(* CODESYS project JobManagement.library
   Company: Bekchoff Automation K.K.
   DocFormat: reStructuredText
   DefaultNamespace: jobmgmt
   Version: 1.0.0.1
   Placeholder: JobManagementFramework
   Author: Takashi Ichihashi
   Title: JobManagementFramework

Project tree, tasks and I/O mapping:
  libraries: Tc2_Standard, * (Beckhoff Automation GmbH); Tc2_System, * (Beckhoff Automation GmbH); Tc2_Utilities, * (Beckhoff Automation GmbH); Tc3_Module, * (Beckhoff Automation GmbH); VisuSymbols, 3.5.10.0 (System)
  DUTs/
    data type ContainerType
    data type E_ErrorId
    data type E_FutureExecutionState
    data type ST_MotionData
  GVLs/
    global variables GVL
    global variables ParamFuturesLib
  POUs/
    model/
      activities/
        function block FB_observer [ST]: subscribe_job_directory, subscribe_job_event
        function block FutureCounterBlink [ST]: abort, counter, error_reset, error_test, execute, init, nErrorID, quit, set_options, set_parameter
        function block FutureCounterBlinkCreator [ST]: create_future, destroy_future, set_options, set_parameter
        function block FutureTimerBlink [ST]: abort, error_reset, error_test, execute, init, nErrorID, quit, set_options, set_parameter
        function block FutureTimerBlinkCreator [ST]: create_future, destroy_future, set_options, set_parameter
      library/
        function block FB_AbstructContainer [ST]: _append_job, _index_generator_, abort, append_job, auto_start, continuous_mode, create_container, create_job, each_executor, error_reset, execute, executor, future_name, init, nErrorID, num_of_jobs, quit, reset, resume, spawn_job, start, state
        function block FB_AbstructFuture [ST]: abort, error_reset, execute, executor, future_name, init, nErrorID, quit, state
        function block FB_BatchJobContainer [ST]: _append_job, _index_generator_, abort, execute, init, quit, resume, start
        function block FB_BatchJobContainerCreator [ST]: create_future, destroy_future
        function block FB_Executor [ST]: abort, busy, children, continuous_mode, create_container, create_future, current_state, done, error_reset, execute, future, future_creator, id, init, job_event_reporter, last_state, nErrorID, parent_executor, persistent_job, quit, ready, reset, resume, start, uid, upstream_aborting
        function block FB_ExecutorTreeSearch [ST]: search, subscriber
        function block FB_ParallelJobContainer [ST]: _append_job, _index_generator_, abort, execute, init, quit, start
        function block FB_ParallelJobContainerCreator [ST]: create_future, destroy_future
        function block FB_ParallelQueueJobContainer [ST]: _append_job, _index_generator_, abort, execute, init, start
        function block FB_ParallelQueueJobContainerCreator [ST]: create_future, destroy_future
        function block FB_QueueJobContainer [ST]: _append_job, _index_generator_, abort, dequeue, execute, init, start
        function block FB_QueueJobContainerCreator [ST]: create_future, destroy_future
        interface InterfaceContainer: _index_generator_, append_job, auto_start, continuous_mode, create_container, create_job, each_executor, num_of_jobs, reset, resume, spawn_job, start
        interface InterfaceFuture: abort, error_reset, execute, executor, future_name, init, nErrorID, quit, state
        interface InterfaceObserver: subscribe_job_directory, subscribe_job_event
        interface InterfaceTaskCreator: create_future, destroy_future
    program MAIN [ST]
  VISUs/
    visualisation Visualization
    visualisation Visualization_1
  text list GlobalTextList
*)

// DUTs/ContainerType
{attribute 'qualified_only'}
{attribute 'strict'}
TYPE ContainerType :
(
	BATCH := 0,
	PARALLEL,
	QUEUE,
	PARALLEL_QUEUE
);
END_TYPE

// DUTs/E_ErrorId
{attribute 'qualified_only'}
{attribute 'strict'}
TYPE E_ErrorId :
(
	PASSIVE_ABORT := 16#FFFFFFFF,
	NOT_CONTAINER := 16#FFFFFFFE
) UDINT;
END_TYPE

// DUTs/E_FutureExecutionState
{attribute 'qualified_only'}
{attribute 'strict'}
{attribute 'to_string'}
TYPE E_FutureExecutionState :
(
	idle := 0,
	init,
	wait_for_process,
	process,
	abort,
	pause,
	quit,
	finish
);
END_TYPE

// DUTs/ST_MotionData
TYPE ST_MotionData :
STRUCT
	name: STRING;
	position: LREAL;
	speed: LREAL;
	accel: LREAL;
END_STRUCT
END_TYPE

// GVLs/GVL
{attribute 'qualified_only'}
VAR_GLOBAL
	batch_job_container_creator : FB_BatchJobContainerCreator;
	parallel_job_container_creator : FB_ParallelJobContainerCreator;
	queue_job_container_creator : FB_QueueJobContainerCreator;
	parallel_queue_job_container_creator : FB_ParallelQueueJobContainerCreator;
END_VAR

// GVLs/ParamFuturesLib
{attribute 'qualified_only'}
VAR_GLOBAL CONSTANT
	MAX_TASK_NUM : UINT := 1000; // Number of max jobs in job container object.
	MAX_STRING_LENGTH : UDINT := 255; // Max string length of task name.
END_VAR

// POUs/model/activities/FB_observer
FUNCTION_BLOCK FB_observer IMPLEMENTS InterfaceObserver
VAR_INPUT
END_VAR
VAR_OUTPUT
	{attribute 'TcEncoding':='UTF-8'}
	text : T_MAXSTRING;
END_VAR
VAR
END_VAR

METHOD subscribe_job_directory : BOOL
VAR_INPUT
	executor	: REFERENCE TO FB_Executor;
END_VAR
VAR
	job_log : STRING;
END_VAR
IF __ISVALIDREF(executor) THEN

	job_log := CONCAT(job_log, 'JOB STRUCTURE');
	IF executor.future <> 0 THEN
		job_log := CONCAT(job_log, '/ FUTURE_NAME : ');
		job_log := CONCAT(job_log, executor.future.future_name);
		job_log := CONCAT(job_log, ', ');	
	END_IF
	job_log := CONCAT(job_log, 'JOB_ID : ');
	job_log := CONCAT(job_log, executor.uid);

	ADSLOGSTR(msgCtrlMask := ADSLOG_MSGTYPE_LOG, msgFmtStr := job_log, strArg := '');
END_IF
END_METHOD

METHOD subscribe_job_event : BOOL
VAR_INPUT
	subject		: T_MaxString;
	old_state	: E_FutureExecutionState;
	new_state	: E_FutureExecutionState;
	record_time	: Tc2_Utilities.T_FILETIME64;
	executor	: REFERENCE TO FB_Executor;
END_VAR
VAR_INST
	fb_timezone_info : FB_GetTimeZoneInformation := (bExecute := TRUE);
END_VAR
VAR
	last_state : STRING;
	current_state : STRING;
	container : InterfaceContainer;
	num_of_jobs : UINT;
END_VAR
last_state := TO_STRING(old_state);
current_state := TO_STRING(new_state);

IF __QUERYINTERFACE(executor.future, container) THEN
	num_of_jobs := container.num_of_jobs;
ELSE
	num_of_jobs := 1;
END_IF


IF __ISVALIDREF(executor) THEN
	fb_timezone_info();
	text := FILETIME64_TO_ISO8601(fileTime := record_time, nBias := DINT_TO_INT(fb_timezone_info.tzInfo.bias), bUTC := TRUE,nPrecision := 6);
	text := CONCAT(text, '	');
	text := CONCAT(text, subject);
	text := CONCAT(text, '	');
	text := CONCAT(text, TO_STRING(current_state));
	text := CONCAT(text, '	');
	text := CONCAT(text, TO_STRING(executor.nErrorID));
	text := CONCAT(text, '		');
	text := CONCAT(text, executor.future.future_name);
	text := CONCAT(text, '		');
	text := CONCAT(text, executor.uid);
	text := CONCAT(text, '		');
	text := CONCAT(text, TO_STRING(num_of_jobs));
	
	
	ADSLOGSTR(msgCtrlMask := ADSLOG_MSGTYPE_LOG,
 			 msgFmtStr := text, 
			strArg := '');	
END_IF

subscribe_job_event := TRUE;
END_METHOD

END_FUNCTION_BLOCK

// POUs/model/library/InterfaceObserver
INTERFACE InterfaceObserver

METHOD subscribe_job_directory : BOOL
VAR_INPUT
	executor: REFERENCE TO FB_Executor; // Represent reference to subscribed job object
END_VAR
END_METHOD

METHOD subscribe_job_event : BOOL
VAR_INPUT
	subject	  : T_MaxString;	// Subject text of event
	old_state : E_FutureExecutionState; // Job state before transition.
	new_state : E_FutureExecutionState; // Job state after transition.
	record_time	: T_FILETIME64; // File-time at the time of transition.
	executor	: REFERENCE TO FB_Executor; // Reference to job instance of which transition occurs.
END_VAR
END_METHOD

END_INTERFACE

// POUs/model/library/FB_Executor
{attribute 'enable_dynamic_creation'}
FUNCTION_BLOCK FB_Executor
VAR_INPUT
END_VAR
VAR_OUTPUT
END_VAR
VAR
	{attribute 'TcEncoding':='UTF-8'}
	_id : T_MaxString;
	_done : BOOL;
	_start : BOOL;
	_resume : BOOL;
	_passive_abort : BOOL;
	_quit : BOOL;
	_upstream_aborting : BOOL := TRUE;
	 {attribute 'TcAnalytics'}
	 _state :E_FutureExecutionState := E_FutureExecutionState.idle;
	_last_state  :E_FutureExecutionState;
	_error_id : UDINT;
	_aborting :BOOL;
	_quitting :BOOL;
	_interface_container : InterfaceContainer := 0;
	_job_event_reporter: InterfaceObserver;
	_future_creator : InterfaceTaskCreator;
	_future : InterfaceFuture;
	_parent_executor : REFERENCE TO FB_Executor REF= 0;
	_persistent_job : BOOL;
END_VAR

(*abort method

*)
METHOD abort : BOOL // Return TRUE if finish.
VAR_INPUT
END_VAR
IF _state = E_FutureExecutionState.init OR
   _state = E_FutureExecutionState.process OR
   _state = E_FutureExecutionState.quit THEN
   	_start := FALSE;
	_passive_abort := TRUE;	
	THIS^.execute();
END_IF

IF 	_passive_abort AND _state = E_FutureExecutionState.abort THEN
	abort := NOT _aborting;
ELSE
	abort := TRUE;
END_IF
END_METHOD

PROPERTY busy : BOOL
GET
busy := (	_state = E_FutureExecutionState.init OR	
			_state = E_FutureExecutionState.process OR 
			_state = E_FutureExecutionState.quit
		);
END_GET
END_PROPERTY

PROPERTY children : InterfaceContainer // Accesser for interface pointer to child container instance.
GET
children := _interface_container;
END_GET
END_PROPERTY

PROPERTY continuous_mode : bool // Make true if keep executing state after all jobs be finished.
SET
IF _future <> 0 THEN
	IF __QUERYINTERFACE(_future, _interface_container) THEN
		_interface_container.continuous_mode := continuous_mode;
	END_IF	
END_IF
END_SET
END_PROPERTY

METHOD create_container : InterfaceContainer // Make container object onto child.
VAR_INPUT
	container_type : ContainerType; // specify container type
	name: STRING;	// specify future name
END_VAR
VAR
	delete_existing_container : BOOL;
	created_future : InterfaceFuture;
END_VAR
IF _interface_container <> 0 THEN
 	IF _interface_container.reset(FALSE) THEN
		delete_existing_container := TRUE;
	ELSE
		delete_existing_container := FALSE;
	END_IF
ELSE
	delete_existing_container := TRUE;
END_IF

IF delete_existing_container THEN
	CASE container_type OF
		ContainerType.BATCH:
			created_future := create_future(GVL.batch_job_container_creator, name);
			created_future.executor.persistent_job := FALSE;
		ContainerType.PARALLEL:
			created_future := create_future(GVL.parallel_job_container_creator, name);
			created_future.executor.persistent_job := FALSE;
		ContainerType.QUEUE:
			created_future := create_future(GVL.queue_job_container_creator, name);
			created_future.executor.persistent_job := TRUE;
		ContainerType.PARALLEL_QUEUE:
			created_future := create_future(GVL.parallel_queue_job_container_creator, name);
			created_future.executor.persistent_job := TRUE;
	END_CASE
	THIS^.init();
	create_container := THIS^.children;
END_IF
END_METHOD

METHOD create_future : InterfaceFuture // Create future dynamically.
VAR_INPUT
	creator : InterfaceTaskCreator; // Specify creator object by which Interface Task Creator implemented.
	future_name: STRING; // Spcfigy future name.
END_VAR
_future_creator := creator;
IF _future_creator <> 0 THEN
	THIS^.future := creator.create_future(future_name);
END_IF
create_future := _future;
END_METHOD

{attribute 'OPC.UA.DA.Property' := '1'}
{attribute 'monitoring' := 'call'}
{attribute 'OPC.UA.DA.Description' := 'Current state of this executor object.'}
PROPERTY current_state : E_FutureExecutionState // Get current job state
GET
current_state := _state;
END_GET
END_PROPERTY

PROPERTY done : BOOL // Present true if process be finished.
GET
done := _done;
END_GET
END_PROPERTY

METHOD error_reset : BOOL
VAR_INPUT
END_VAR
IF _future <> 0 THEN
	IF _future.error_reset() THEN
		error_reset := TRUE;
		IF _job_event_reporter <> 0 THEN
			_job_event_reporter.subscribe_job_event(
						subject := 'ERROR_RESET',
						old_state := _last_state,
						new_state := _state,
						record_time := F_GetSystemTime(),
						executor := THIS^
				);
		END_IF
	ELSE
		error_reset := FALSE;
	END_IF
	_error_id := _future.nErrorID;
ELSE
	_error_id := 0;
	error_reset := TRUE;
END_IF
END_METHOD

METHOD execute : BOOL // Execute future process and return TRUE if all task are finished.
VAR_INST
	_state_mem :E_FutureExecutionState;
	_logging :BOOL;
	delay : TIME := T#3S;
	sleep : TON;
END_VAR
VAR
	_executor : REFERENCE TO FB_Executor;
	start_all_children : BOOL;
	exe: INT;
END_VAR
IF _future = 0 THEN
	execute := TRUE;
	RETURN;
ELSE
	execute := FALSE;
END_IF

IF _passive_abort THEN
	_state := E_FutureExecutionState.abort;
	IF _error_id = 0 THEN
		_error_id := E_ErrorId.PASSIVE_ABORT;
	END_IF
	_passive_abort := FALSE;
END_IF

IF _quit THEN
	_state := E_FutureExecutionState.quit;
END_IF
_quit := FALSE;

CASE _state OF
	E_FutureExecutionState.idle:
		ADSLOGSTR(msgCtrlMask := ADSLOG_MSGTYPE_LOG, msgFmtStr := TO_STRING(_future.state), strArg := '');
		IF _future.state = E_FutureExecutionState.idle OR 
			_future.state = E_FutureExecutionState.finish THEN
			IF init() THEN
				_state := E_FutureExecutionState.init;
			END_IF
		END_IF
	E_FutureExecutionState.init:
		IF _future.init() THEN
			IF _future.nErrorID = 0 THEN
				_state := E_FutureExecutionState.wait_for_process;
			ELSE
				_last_state := E_FutureExecutionState.init;
				_error_id := _future.nErrorID;
				_state := E_FutureExecutionState.abort;
			END_IF
		END_IF
	E_FutureExecutionState.wait_for_process: 
		IF _start THEN
			_state := E_FutureExecutionState.process;
			_start := FALSE;
		END_IF
	E_FutureExecutionState.process: 
		IF _future.execute() THEN
			IF _future.nErrorID = 0 THEN
				_state := E_FutureExecutionState.quit;
				_done := TRUE;
			ELSE
				_error_id := _future.nErrorID;
				_state := E_FutureExecutionState.abort;
			END_IF
		END_IF
	E_FutureExecutionState.abort:
		IF _aborting THEN
			_resume := FALSE;
			IF _upstream_aborting AND __ISVALIDREF(_parent_executor) THEN
				_parent_executor.abort();				
			END_IF
			IF _future.abort() THEN
				_aborting := FALSE;
			END_IF
		ELSIF _resume THEN
			_state := _last_state;
			IF _error_id = E_ErrorId.PASSIVE_ABORT THEN
				_error_id := 0;
			END_IF
			_resume := FALSE;
		END_IF
	E_FutureExecutionState.quit:
		IF _future.quit() THEN
			IF _future.nErrorID = 0 THEN
				_state := E_FutureExecutionState.finish;
			ELSE
				_error_id := _future.nErrorID;
				_state := E_FutureExecutionState.abort;
			END_IF
			_quitting := FALSE;
		END_IF
	E_FutureExecutionState.finish:
		IF NOT _logging THEN
			execute := TRUE;
		END_IF
END_CASE

IF _state <> _state_mem THEN
	_last_state := _state_mem;

	IF _state = E_FutureExecutionState.init OR
		_state = E_FutureExecutionState.process OR
		_state = E_FutureExecutionState.quit THEN
		_error_id := 0;
	END_IF

	IF _state = E_FutureExecutionState.abort THEN
		_aborting := TRUE;
	END_IF
	
	IF _state = E_FutureExecutionState.quit THEN
		sleep(IN := FALSE);
		_quitting := TRUE;
	END_IF
		
	IF _job_event_reporter <> 0 AND _state >= E_FutureExecutionState.idle AND _state <= E_FutureExecutionState.finish THEN
		// reporter
		_logging := TRUE;
	END_IF
END_IF

_state_mem := _state;

IF _logging THEN
	IF _job_event_reporter.subscribe_job_event(
			subject := 'TRANSITION',
			old_state := _last_state,
			new_state := _state,
			record_time := F_GetSystemTime(),
			executor := THIS^
	) THEN
		_logging := FALSE;
	END_IF
END_IF

IF _future <> 0 THEN
	_future.state := _state;
END_IF
END_METHOD

PROPERTY future : InterfaceFuture // Set future instance direct.
GET
future := _future;
END_GET
SET
_future := future;
_future.state := _state;
_future.executor REF= THIS^;
IF NOT __QUERYINTERFACE(_future, _interface_container) THEN
	_interface_container := 0;
END_IF
END_SET
END_PROPERTY

PROPERTY future_creator : InterfaceTaskCreator // Set creator instance.
SET
_future_creator := future_creator;
END_SET
END_PROPERTY

PROPERTY id : T_MaxString // Get job id.
GET
id := _id;
END_GET
SET
_id := id;
END_SET
END_PROPERTY

METHOD init : BOOL // Return TRUE if finish.
VAR_INPUT
END_VAR
_done := FALSE;
_passive_abort := FALSE;
_start := FALSE;
_state := E_FutureExecutionState.init;
_error_id := 0;
IF _future <> 0 THEN
	_future.init();
END_IF

INIT := TRUE;
END_METHOD

PROPERTY job_event_reporter : InterfaceObserver
GET
job_event_reporter := _job_event_reporter;
END_GET
SET
VAR
	executor :REFERENCE TO FB_Executor;
END_VAR
_job_event_reporter := job_event_reporter;
IF THIS^.children <> 0 THEN
	REPEAT
		executor REF= THIS^.children.each_executor;
		IF __ISVALIDREF(executor) THEN
			executor.job_event_reporter := job_event_reporter;
		END_IF
	UNTIL
		NOT __ISVALIDREF(executor)
	END_REPEAT
END_IF
END_SET
END_PROPERTY

PROPERTY last_state : E_FutureExecutionState
GET
last_state := _last_state;
END_GET
END_PROPERTY

PROPERTY nErrorID : UDINT // Present error code when each process,init(), execute(), quit() are finished. '0' represent normal condition without any errors.
GET
nErrorID := _error_id;
END_GET
END_PROPERTY

PROPERTY parent_executor : REFERENCE TO FB_Executor
GET
parent_executor REF= _parent_executor;
END_GET
SET
_parent_executor REF= parent_executor;
END_SET
END_PROPERTY

PROPERTY persistent_job : BOOL
GET
persistent_job := _persistent_job;
END_GET
SET
_persistent_job := persistent_job;
END_SET
END_PROPERTY

METHOD quit : BOOL // Return TRUE if finish.
VAR_INPUT
END_VAR
IF _state = E_FutureExecutionState.init OR
   _state = E_FutureExecutionState.process OR
   _state = E_FutureExecutionState.quit THEN
	_quit := TRUE;	
END_IF

IF 	_quit AND _state = E_FutureExecutionState.quit THEN
	quit := NOT _quitting;
ELSE
	quit := TRUE;
END_IF
END_METHOD

PROPERTY ready : BOOL
GET
ready := _state = E_FutureExecutionState.wait_for_process;
END_GET
END_PROPERTY

METHOD reset : BOOL // Return TRUE if finish.
VAR_INPUT
	deep : BOOL := FALSE;
END_VAR
VAR
	_reset_children :BOOL := FALSE;
END_VAR
// Waiting finish process and remove jobs from container items.
IF THIS^.busy THEN
	THIS^.abort();
ELSIF _interface_container <> 0 AND ( NOT _persistent_job OR deep) THEN
	IF _interface_container.reset(deep) THEN
		_reset_children := TRUE;
	END_IF
ELSE
	_reset_children := TRUE;
END_IF

// Remove my future.
IF _reset_children AND _future <> 0 THEN
	IF  NOT _persistent_job OR deep THEN
		IF _future_creator <> 0 THEN
			_future := _future_creator.destroy_future(_future);
		ELSIF _future.init() THEN
			_future.state := E_FutureExecutionState.idle;
			_future := 0;
		END_IF
		IF _future = 0 THEN
			_interface_container := 0;
			reset := TRUE;
		END_IF
	ELSE
		IF _future.init() THEN
			reset := TRUE;
		END_IF
	END_IF
END_IF
END_METHOD

METHOD resume : BOOL
VAR_INST
	_executor : REFERENCE TO FB_Executor;
END_VAR
_resume := TRUE;
IF _interface_container <> 0 THEN
	IF NOT _interface_container.resume() THEN
		_resume := FALSE;
	END_IF
END_IF
IF NOT _resume THEN
	_future.execute();
END_IF
resume := _resume;
END_METHOD

METHOD start : BOOL
VAR
	_start_children :BOOL := FALSE;
END_VAR
// Send start signal to children.
IF _interface_container <> 0 THEN
	IF _interface_container.start() THEN
		_start_children := TRUE;
	END_IF
ELSE
	_start_children := TRUE;
END_IF

// Start my future.
IF _start_children THEN
	_start := _state = E_FutureExecutionState.wait_for_process;
	start := TRUE;
END_IF
END_METHOD

PROPERTY uid : T_MaxString
GET
VAR
	_eval_executor : REFERENCE TO FB_Executor;
	_uid : T_MaxString;
END_VAR
_eval_executor REF= _parent_executor;
_uid := _id;
REPEAT
	_uid := CONCAT('/',_uid);
	IF __ISVALIDREF(_eval_executor) THEN
		_uid := CONCAT(_eval_executor.id, _uid);
		_eval_executor REF= _eval_executor._parent_executor;
	END_IF
UNTIL
	NOT __ISVALIDREF(_eval_executor)
END_REPEAT

uid := _uid;
END_GET
END_PROPERTY

PROPERTY upstream_aborting : BOOL
GET
upstream_aborting := _upstream_aborting;
END_GET
SET
_upstream_aborting := upstream_aborting;
END_SET
END_PROPERTY

END_FUNCTION_BLOCK

// POUs/model/library/InterfaceContainer
INTERFACE InterfaceContainer EXTENDS __SYSTEM.IQueryInterface

(* This is the generator that iteratively generates references to FB_executor instances*)
METHOD _index_generator_ : UINT;
VAR_INPUT
END_VAR
END_METHOD

METHOD append_job : BOOL
VAR_INPUT
	executor	: REFERENCE TO FB_Executor;
END_VAR
END_METHOD

PROPERTY auto_start : bool
SET
END_SET
END_PROPERTY

PROPERTY continuous_mode : bool
SET
END_SET
END_PROPERTY

METHOD create_container : REFERENCE TO FB_Executor
VAR_INPUT
	container_type : ContainerType;
	name: STRING;
END_VAR
END_METHOD

METHOD create_job : REFERENCE TO FB_Executor
VAR_INPUT
	creator : InterfaceTaskCreator;
	future_name: STRING;
END_VAR
END_METHOD

PROPERTY each_executor : REFERENCE TO FB_Executor
GET
END_GET
END_PROPERTY

PROPERTY num_of_jobs : UINT
GET
END_GET
END_PROPERTY

METHOD reset : BOOL // Return TRUE if finish.
VAR_INPUT
	deep : BOOL := FALSE;
END_VAR
END_METHOD

METHOD resume : BOOL
VAR_INPUT
END_VAR
END_METHOD

METHOD spawn_job : REFERENCE TO FB_Executor
VAR_INPUT
	future : InterfaceFuture;
END_VAR
END_METHOD

METHOD start : BOOL
END_METHOD

END_INTERFACE

// POUs/model/library/InterfaceTaskCreator
INTERFACE InterfaceTaskCreator

METHOD create_future : InterfaceFuture
VAR_INPUT
	future_name :STRING; // Specify future name
END_VAR
END_METHOD

METHOD destroy_future : InterfaceFuture
VAR_INPUT
	future : InterfaceFuture; // Specify future instance whtat you want to delete.
END_VAR
END_METHOD

END_INTERFACE

// POUs/model/library/InterfaceFuture
{attribute 'enable_dynamic_creation'}
INTERFACE InterfaceFuture EXTENDS __System.IQueryInterface

METHOD abort : BOOL // Return TRUE if finish.
VAR_INPUT
END_VAR
END_METHOD

METHOD error_reset : BOOL
VAR_INPUT
END_VAR
END_METHOD

METHOD execute : BOOL // Return TRUE if finish.
VAR_INPUT
END_VAR
END_METHOD

PROPERTY executor : REFERENCE TO FB_Executor
GET
END_GET
SET
END_SET
END_PROPERTY

PROPERTY future_name : STRING // Name of future.
GET
END_GET
SET
END_SET
END_PROPERTY

METHOD init : BOOL // Return TRUE if finish.
VAR_INPUT
END_VAR
END_METHOD

PROPERTY nErrorID : UDINT // Set result code when finished any method. 0 should be set when normal case.
GET
END_GET
END_PROPERTY

METHOD quit : BOOL // Return TRUE if finish.
VAR_INPUT
END_VAR
END_METHOD

PROPERTY state : E_FutureExecutionState // Execution state of this future.
GET
END_GET
SET
END_SET
END_PROPERTY

END_INTERFACE

// POUs/model/activities/FutureCounterBlink
{attribute 'enable_dynamic_creation'}
FUNCTION_BLOCK FutureCounterBlink EXTENDS FB_AbstructFuture
VAR_INPUT
END_VAR
VAR_OUTPUT
END_VAR
VAR
	process_timer: TON;
	blink_timer: TON;
	_counter :UINT;
	_error_id :UDINT;
	_target_count: UINT;
	_count_trigger: REFERENCE TO BOOL;
	_output: REFERENCE TO BOOL;
	_error_test :BOOL;
END_VAR

METHOD abort : BOOL
// The warning can be disabled here as the user is aware of the risk that the reference may not be valid by checking its validity
{warning disable C0371}
// Checking the VAR_IN_OUT reference, leave the current method in case of invalid reference
IF NOT __ISVALIDREF(_output) THEN
     RETURN;
END_IF

_output := FALSE;
abort := TRUE;

// The warning may be restored at the end of the access area
{warning restore C0371}
END_METHOD

PROPERTY counter : UINT
GET
counter := _counter;
END_GET
END_PROPERTY

METHOD error_reset : BOOL // Must be overrided if future has any errors.
_error_test := FALSE;
_error_id := 0;
error_reset := TRUE;
END_METHOD

PROPERTY error_test : BOOL
SET
_error_test := error_test;
END_SET
END_PROPERTY

METHOD execute : BOOL
VAR_INPUT
END_VAR
VAR_INST
	input_memory :BOOL;
END_VAR
// The warning can be disabled here as the user is aware of the risk that the reference may not be valid by checking its validity
{warning disable C0371}
// Checking the VAR_IN_OUT reference, leave the current method in case of invalid reference
IF NOT __ISVALIDREF(_output) OR NOT __ISVALIDREF(_count_trigger) THEN
	_error_id := 1;
     RETURN;
END_IF

IF _error_test THEN
	_error_id := 9;
	execute := TRUE;
END_IF

_output := TRUE;
IF _count_trigger AND NOT input_memory THEN
	_counter := _counter + 1;
END_IF
input_memory := _count_trigger;
IF _counter > _target_count THEN
	execute := TRUE;
END_IF

// The warning may be restored at the end of the access area
{warning restore C0371}
END_METHOD

METHOD init : BOOL
VAR_INPUT
END_VAR
// The warning can be disabled here as the user is aware of the risk that the reference may not be valid by checking its validity
{warning disable C0371}
// Checking the VAR_IN_OUT reference, leave the current method in case of invalid reference
IF NOT __ISVALIDREF(_output) THEN
	_error_id := 1;
     RETURN;
END_IF

_output := FALSE;
process_timer(IN := FALSE);
blink_timer(IN := FALSE);
_counter := 0;
init := TRUE;

// The warning may be restored at the end of the access area
{warning restore C0371}
END_METHOD

PROPERTY nErrorID : UDINT
GET
nErrorID := _error_id;
END_GET
END_PROPERTY

METHOD quit : BOOL
THIS^.init();
quit := TRUE;
END_METHOD

METHOD set_options : BOOL
VAR_INPUT
	error_test: BOOL;
END_VAR
_error_test := error_test;
END_METHOD

METHOD set_parameter : BOOL
VAR_INPUT
	target_count: UINT;
	count_trigger : REFERENCE TO BOOL;
	output		: REFERENCE TO BOOL;
END_VAR
_count_trigger REF= count_trigger;
_output REF= output;
_target_count := target_count;
END_METHOD

END_FUNCTION_BLOCK

// POUs/model/library/FB_AbstructFuture
FUNCTION_BLOCK ABSTRACT FB_AbstructFuture IMPLEMENTS InterfaceFuture
VAR_INPUT
END_VAR
VAR_OUTPUT
END_VAR
VAR
	_executor : REFERENCE TO FB_Executor;
	{attribute 'TcEncoding':='UTF-8'}
	_future_name :STRING := 'NO_NAME';
	_busy : BOOL; 
	_state : E_FutureExecutionState;
END_VAR

METHOD abort : BOOL // Must be overrided if future has any errors.
abort := TRUE;
END_METHOD

METHOD error_reset : BOOL // Must be overrided if future has any errors.
error_reset := TRUE;
END_METHOD

METHOD execute : BOOL // Must be overrided.
END_METHOD

PROPERTY executor : REFERENCE TO FB_Executor
GET
executor REF= _executor;
END_GET
SET
_executor REF= executor;
END_SET
END_PROPERTY

PROPERTY future_name : STRING // Name of future.
GET
future_name := _future_name;
END_GET
SET
_future_name := future_name;
END_SET
END_PROPERTY

METHOD init : BOOL // Return TRUE if finish.
init := TRUE;
END_METHOD

PROPERTY nErrorID : UDINT // Must be overrided if future has any errors.
GET
END_GET
END_PROPERTY

METHOD quit : BOOL // Return TRUE if finish.
init();
quit := TRUE;
END_METHOD

PROPERTY state : E_FutureExecutionState // Execution state of this future.
GET
state := _state;
END_GET
SET
_state := state;
END_SET
END_PROPERTY

END_FUNCTION_BLOCK

// POUs/model/activities/FutureCounterBlinkCreator
FUNCTION_BLOCK FutureCounterBlinkCreator IMPLEMENTS InterfaceTaskCreator
VAR_INPUT
END_VAR
VAR_OUTPUT
END_VAR
VAR
	_target_count: UINT;
	_count_trigger: REFERENCE TO BOOL;
	_output: REFERENCE TO BOOL;
	_error_test :BOOL;
END_VAR

{warning 'add method implementation '}
METHOD create_future : InterfaceFuture
VAR_INPUT
	future_name :STRING;
END_VAR
VAR
	_p_future : POINTER TO FutureCounterBlink;
END_VAR
_p_future := __NEW(FutureCounterBlink);
_p_future^.future_name := future_name;
_p_future^.set_parameter(_target_count, _count_trigger, _output);
_p_future^.error_test := _error_test;
create_future := _p_future^;
END_METHOD

{warning 'add method implementation '}
METHOD destroy_future : InterfaceFuture
VAR_INPUT
	future : InterfaceFuture;
END_VAR
VAR
	_p_future : POINTER TO FutureCounterBlink;
END_VAR
IF __QUERYPOINTER(future, _p_future) THEN
	__DELETE(_p_future);
	IF _p_future = 0  THEN
		destroy_future := 0;
	END_IF
END_IF
END_METHOD

METHOD set_options : BOOL
VAR_INPUT
	error_test: BOOL;
END_VAR
_error_test := error_test;
END_METHOD

METHOD set_parameter : BOOL
VAR_INPUT
	target_count: UINT;
	count_trigger : REFERENCE TO BOOL;
	output		: REFERENCE TO BOOL;
END_VAR
_count_trigger REF= count_trigger;
_output REF= output;
_target_count := target_count;
END_METHOD

END_FUNCTION_BLOCK

// POUs/model/activities/FutureTimerBlink
{attribute 'enable_dynamic_creation'}
FUNCTION_BLOCK FutureTimerBlink EXTENDS FB_AbstructFuture
VAR_INPUT
END_VAR
VAR_OUTPUT
END_VAR
VAR
	process_timer: TON;
	blink_timer: TON;
	_set_time :TIME;
	_result :UDINT;
	_output: REFERENCE TO BOOL;
	_process_time: TIME;
	_error_test :BOOL;
END_VAR

METHOD abort : BOOL
IF process_timer.IN THEN
	_set_time := process_timer.PT - process_timer.ET;
END_IF
process_timer(IN := FALSE);
_output := FALSE;
abort := TRUE;
END_METHOD

METHOD error_reset : BOOL // Must be overrided if future has any errors.
_error_test := FALSE;
_result := 0;
error_reset := TRUE;
END_METHOD

PROPERTY error_test : BOOL
SET
_error_test := error_test;
END_SET
END_PROPERTY

METHOD execute : BOOL
VAR_INPUT
END_VAR
blink_timer(IN := NOT blink_timer.Q, PT := T#0.5S);
IF _output AND blink_timer.Q THEN
	_output := FALSE;
ELSIF blink_timer.Q THEN
	_output := TRUE;
END_IF
process_timer(IN := TRUE,PT := _process_time);
execute := process_timer.Q;

IF _error_test THEN
	_result := 9;
	execute := TRUE;
END_IF
END_METHOD

METHOD init : BOOL
VAR_INPUT
END_VAR
_output := FALSE;
_set_time := _process_time;
process_timer(IN := FALSE);
blink_timer(IN := FALSE);
init := TRUE;
END_METHOD

PROPERTY nErrorID : UDINT
GET
END_GET
END_PROPERTY

METHOD quit : BOOL
THIS^.init();
quit := TRUE;
END_METHOD

METHOD set_options : BOOL
VAR_INPUT
	error_test: BOOL;
END_VAR
_error_test := error_test;
END_METHOD

METHOD set_parameter : BOOL
VAR_INPUT
	process_time: TIME;
	output		: REFERENCE TO BOOL;
END_VAR
_process_time := process_time;
_output REF= output;
END_METHOD

END_FUNCTION_BLOCK

// POUs/model/activities/FutureTimerBlinkCreator
FUNCTION_BLOCK FutureTimerBlinkCreator IMPLEMENTS InterfaceTaskCreator
VAR_INPUT
END_VAR
VAR_OUTPUT
END_VAR
VAR
	_output: REFERENCE TO BOOL;
	_process_time: TIME;
	_error_test :BOOL;
END_VAR

{warning 'add method implementation '}
METHOD create_future : InterfaceFuture
VAR_INPUT
	future_name	: STRING;
END_VAR
VAR
	_p_future : POINTER TO FutureTimerBlink;
END_VAR
_p_future := __NEW(FutureTimerBlink);
_p_future^.future_name := future_name;
_p_future^.set_parameter(_process_time, _output);
_p_future^.set_options(_error_test);
create_future := _p_future^;
END_METHOD

{warning 'add method implementation '}
METHOD destroy_future : InterfaceFuture
VAR_INPUT
	future	: InterfaceFuture;
END_VAR
VAR
	_p_future : POINTER TO FutureTimerBlink;
END_VAR
IF __QUERYPOINTER(future, _p_future) THEN
	__DELETE(_p_future);
	IF _p_future = 0  THEN
		destroy_future := 0;
	END_IF
END_IF
END_METHOD

METHOD set_options : BOOL
VAR_INPUT
	error_test: BOOL;
END_VAR
_error_test := error_test;
END_METHOD

METHOD set_parameter : BOOL
VAR_INPUT
	process_time: TIME;
	output		: REFERENCE TO BOOL;
END_VAR
_process_time := process_time;
_output REF= output;
END_METHOD

END_FUNCTION_BLOCK

// POUs/model/library/FB_AbstructContainer
FUNCTION_BLOCK ABSTRACT FB_AbstructContainer IMPLEMENTS InterfaceFuture, InterfaceContainer
VAR_INPUT
END_VAR
VAR_OUTPUT
END_VAR
VAR
	_executor : REFERENCE TO FB_Executor;
	{attribute 'TcEncoding':='UTF-8'}
	_name 	: STRING := 'BATCH JOB';
	_executors : ARRAY [1..ParamFuturesLib.MAX_TASK_NUM] OF POINTER TO FB_Executor;
	_auto_start : BOOL := TRUE;
	_start :BOOL;
	_abort : BOOL;
	_num_of_jobs: UINT;
	current_executing_future_id : UINT;
	current_executing_future : InterfaceFuture;
	_continuous_mode : BOOL;
	_error_id :UDINT;
	_state :E_FutureExecutionState;
	_job_event_reporter : InterfaceObserver;
END_VAR

METHOD PROTECTED _append_job : BOOL
VAR_INPUT
	executor	: REFERENCE TO FB_Executor;
END_VAR
END_METHOD

(* This is the generator that iteratively generates references to FB_executor instances*)
METHOD _index_generator_ : UINT
VAR_INST
	_index : UINT;
END_VAR
_index := _index + 1;
IF _index > _num_of_jobs THEN
	_index := 0;
END_IF
_index_generator_ := _index;
END_METHOD

METHOD abort : BOOL // Return TRUE if finish.
abort := _executors[current_executing_future_id]^.abort();
END_METHOD

{warning 'add method implementation '}
METHOD append_job : BOOL
VAR_INPUT
	executor	: REFERENCE TO FB_Executor;
END_VAR
executor.persistent_job := TRUE;
THIS^._append_job(executor);
END_METHOD

PROPERTY auto_start : BOOL
SET
_auto_start := auto_start;
END_SET
END_PROPERTY

PROPERTY continuous_mode : BOOL
SET
VAR
	_executor : REFERENCE TO FB_Executor;
END_VAR
_continuous_mode := continuous_mode;
REPEAT
	_executor REF= THIS^.each_executor;
	IF __ISVALIDREF(_executor) THEN
		_executor.continuous_mode := continuous_mode;
	END_IF
UNTIL
	NOT __ISVALIDREF(_executor)
END_REPEAT
END_SET
END_PROPERTY

METHOD create_container : REFERENCE TO FB_Executor
VAR_INPUT
	container_type	: ContainerType;
	name	: STRING;
END_VAR
CASE container_type OF
	ContainerType.BATCH:
		create_container REF= THIS^.create_job(GVL.batch_job_container_creator,name);
	ContainerType.PARALLEL:
		create_container REF= THIS^.create_job(GVL.parallel_job_container_creator,name);
	ContainerType.QUEUE:
		create_container REF= THIS^.create_job(GVL.queue_job_container_creator,name);
	ContainerType.PARALLEL_QUEUE:
		create_container REF= THIS^.create_job(GVL.parallel_queue_job_container_creator,name);
END_CASE
END_METHOD

METHOD create_job : REFERENCE TO FB_Executor
VAR_INPUT
	creator	: InterfaceTaskCreator;
	future_name	: STRING;
END_VAR
VAR
	future : InterfaceFuture;
END_VAR
IF _num_of_jobs < ParamFuturesLib.MAX_TASK_NUM THEN
	future := creator.create_future(future_name);
	create_job REF= THIS^.spawn_job(future);
	IF __ISVALIDREF(create_job) THEN
		create_job.future_creator := creator;
	ELSE
		creator.destroy_future(future);
	END_IF
END_IF
END_METHOD

PROPERTY each_executor : REFERENCE TO FB_Executor
GET
VAR
	_index : UINT;
END_VAR
_index := _index_generator_();
IF _index > 0 THEN
	IF _executors[_index] <> 0 THEN
		IF _executors[_index] <> 0 THEN
			each_executor REF= _executors[_index]^;
		ELSE
			each_executor REF= 0;
		END_IF
	END_IF
ELSE
	each_executor REF= 0;
END_IF
END_GET
END_PROPERTY

METHOD error_reset : BOOL
VAR
	_executor : REFERENCE TO FB_Executor;
	complete : BOOL;
END_VAR
complete := TRUE;
REPEAT
	_executor REF= each_executor;
	IF __ISVALIDREF(_executor) THEN
		IF NOT _executor.error_reset() THEN
			complete := FALSE;
		END_IF
	END_IF
UNTIL
	NOT __ISVALIDREF(_executor)
END_REPEAT
IF complete THEN
	_error_id := 0;
END_IF
error_reset := complete;
END_METHOD

METHOD execute : BOOL // Return TRUE if finish.
END_METHOD

PROPERTY executor : REFERENCE TO FB_Executor
GET
executor REF= _executor;
END_GET
SET
_executor REF= executor;
END_SET
END_PROPERTY

PROPERTY future_name : STRING// Name of future.
GET
future_name := _name;
END_GET
SET
_name := future_name;
END_SET
END_PROPERTY

METHOD init : BOOL // Return TRUE if finish.
VAR
	_executor : REFERENCE TO FB_Executor;
	_init_done : BOOL;
END_VAR
_init_done := TRUE;
REPEAT
	_executor REF= THIS^.each_executor;
	IF __ISVALIDREF(_executor) THEN
		_executor.job_event_reporter := _executor.job_event_reporter;
		IF NOT _executor.init() THEN
			_init_done := FALSE;
		END_IF
	END_IF
UNTIL
	NOT __ISVALIDREF(_executor)
END_REPEAT

current_executing_future_id := 1;
_error_id := 0;
init := _init_done;
END_METHOD

PROPERTY nErrorID : UDINT
GET
nErrorID := _error_id;
END_GET
END_PROPERTY

PROPERTY num_of_jobs : UINT
GET
num_of_jobs := _num_of_jobs;
END_GET
END_PROPERTY

METHOD quit : BOOL // Return TRUE if finish.
quit := TRUE;
END_METHOD

METHOD reset : BOOL // Return TRUE if finish.
VAR_INPUT
	deep : BOOL := FALSE;
END_VAR
VAR
	i : UINT;
	_delete_counter : UINT;
	text : STRING;
END_VAR
_delete_counter := 0;
REPEAT
	i := _index_generator_();
	IF _num_of_jobs >= i AND i > 0 THEN
		IF _executors[i] <> 0 THEN
			IF _executors[i]^.reset(deep) THEN
				__DELETE(_executors[i]);
				_delete_counter := _delete_counter + 1;
			END_IF
		END_IF
	END_IF
UNTIL
	i = 0
END_REPEAT
_num_of_jobs := _num_of_jobs - _delete_counter;
reset := _num_of_jobs = 0;
END_METHOD

METHOD resume : BOOL
VAR
	_all_done : BOOL;
END_VAR
VAR_INST
	_executor : REFERENCE TO FB_Executor;
END_VAR
_all_done := TRUE;
REPEAT
	_executor REF= THIS^.each_executor;
	IF __ISVALIDREF(_executor) THEN
		IF NOT _executor.resume() THEN
			_all_done := FALSE;
		END_IF
	END_IF
UNTIL
	NOT __ISVALIDREF(_executor)
END_REPEAT
resume := _all_done;
END_METHOD

METHOD spawn_job : REFERENCE TO FB_Executor
VAR_INPUT
	future : InterfaceFuture;
END_VAR
VAR
	_spawned_executor : POINTER TO FB_Executor;
END_VAR
IF future <> 0 THEN
	_spawned_executor := __NEW(FB_Executor);
	_spawned_executor^.future := future;
	_spawned_executor^.persistent_job := FALSE;
	_append_job(_spawned_executor^);
	spawn_job REF= _spawned_executor^;
ELSE
	spawn_job REF= 0;
END_IF
END_METHOD

METHOD start : BOOL
start := _executors[current_executing_future_id]^.start();
END_METHOD

PROPERTY state : E_FutureExecutionState
GET
state := _state;
END_GET
SET
_state := state;
END_SET
END_PROPERTY

END_FUNCTION_BLOCK

// POUs/model/library/FB_BatchJobContainer
{attribute 'enable_dynamic_creation'}
FUNCTION_BLOCK FB_BatchJobContainer EXTENDS FB_AbstructContainer
VAR_INPUT
END_VAR
VAR_OUTPUT
END_VAR
VAR
	_all_abort : BOOL;
END_VAR

METHOD PROTECTED _append_job : BOOL
VAR_INPUT
	executor	: REFERENCE TO FB_Executor;
END_VAR
VAR
	_parent_future_id: STRING;	
END_VAR
IF __ISVALIDREF(executor) AND _num_of_jobs < ParamFuturesLib.MAX_TASK_NUM THEN
	executor.init();
	_num_of_jobs := _num_of_jobs + 1;
	executor.id := UINT_TO_STRING(_num_of_jobs);
	_executors[_num_of_jobs] := ADR(executor);
	IF  __ISVALIDREF(_executor) THEN
		// Propergate task creator object
		_executors[_num_of_jobs]^.job_event_reporter := _executor.job_event_reporter;
		_executors[_num_of_jobs]^.parent_executor REF= _executor;
		_executors[_num_of_jobs]^.upstream_aborting := _executor.upstream_aborting;
		_parent_future_id := _executor.id;
	END_IF
END_IF
END_METHOD

(* This is the generator that iteratively generates references to FB_executor instances*)
METHOD _index_generator_ : UINT
VAR_INST
	_index : UINT;
END_VAR
_index := _index + 1;
IF _index > _num_of_jobs THEN
	_index := 0;
END_IF
_index_generator_ := _index;
END_METHOD

METHOD abort : BOOL // Return TRUE if finish.
abort := _executors[current_executing_future_id]^.abort();
END_METHOD

METHOD execute : BOOL // Return TRUE if finish.
VAR_INST
	i :UINT;
	complete_last_proess :BOOL;
	complete_all_process :BOOL;
END_VAR
IF _num_of_jobs = 0 THEN
	RETURN;
END_IF



FOR i := 1 TO _num_of_jobs DO
	complete_all_process := _executors[i]^.execute();
	_error_id := _executors[i]^.nErrorID;
END_FOR

IF current_executing_future_id > 1 THEN
	complete_last_proess := _executors[current_executing_future_id - 1]^.done;
ELSE
	complete_last_proess := TRUE;
END_IF

CASE _executors[current_executing_future_id]^.current_state OF
	E_FutureExecutionState.init, E_FutureExecutionState.process, E_FutureExecutionState.quit:
		_all_abort := FALSE;
		IF _abort THEN
			IF _executors[current_executing_future_id]^.abort() THEN
				_all_abort := TRUE;
			END_IF
		END_IF
	E_FutureExecutionState.wait_for_process:
		IF _executors[current_executing_future_id]^.ready AND complete_last_proess AND _auto_start THEN
			_executors[current_executing_future_id]^.start();
		END_IF
END_CASE

IF complete_all_process THEN
	execute := NOT _continuous_mode;
ELSIF _executors[current_executing_future_id]^.done AND current_executing_future_id < _num_of_jobs THEN
	execute := FALSE;
	current_executing_future_id := current_executing_future_id + 1;
END_IF

current_executing_future := _executors[current_executing_future_id]^.future;
END_METHOD

METHOD init : BOOL // Return TRUE if finish.
VAR
	_executor : REFERENCE TO FB_Executor;
	_init_done : BOOL;
END_VAR
_init_done := TRUE;
REPEAT
	_executor REF= THIS^.each_executor;
	IF __ISVALIDREF(_executor) THEN
		_executor.job_event_reporter := _executor.job_event_reporter;
		IF NOT _executor.init() THEN
			_init_done := FALSE;
		END_IF
	END_IF
UNTIL
	NOT __ISVALIDREF(_executor)
END_REPEAT

current_executing_future_id := 1;
_error_id := 0;
init := _init_done;
END_METHOD

METHOD quit : BOOL // Return TRUE if finish.
VAR_INST
	i: UINT;
	complete_all_task :BOOL;
END_VAR
complete_all_task := TRUE;
FOR i := 1 TO _num_of_jobs DO
	_executors[i]^.execute();
	IF NOT (_executors[i]^.current_state = E_FutureExecutionState.finish) THEN
		complete_all_task := FALSE;	
	END_IF
END_FOR
IF complete_all_task THEN
	current_executing_future_id := 0;
	quit := TRUE;
ELSE
	quit := FALSE;
END_IF
END_METHOD

METHOD resume : BOOL
resume := _executors[current_executing_future_id]^.resume();
END_METHOD

METHOD start : BOOL
start := _executors[current_executing_future_id]^.start();
END_METHOD

END_FUNCTION_BLOCK

// POUs/model/library/FB_BatchJobContainerCreator
FUNCTION_BLOCK FB_BatchJobContainerCreator IMPLEMENTS InterfaceTaskCreator
VAR_INPUT
END_VAR
VAR_OUTPUT
END_VAR
VAR
END_VAR

METHOD create_future : InterfaceFuture
VAR_INPUT
	future_name :STRING;
END_VAR
VAR
	_p_future : POINTER TO FB_BatchJobContainer;
END_VAR
_p_future := __NEW(FB_BatchJobContainer);
_p_future^.future_name := future_name;
create_future := _p_future^;
END_METHOD

{warning 'add method implementation '}
METHOD destroy_future : InterfaceFuture
VAR_INPUT
	future	: InterfaceFuture;
END_VAR
VAR
	_p_future : POINTER TO FB_BatchJobContainer;
END_VAR
IF __QUERYPOINTER(future, _p_future) THEN
	__DELETE(_p_future);
	IF _p_future = 0  THEN
		destroy_future := 0;
	END_IF
END_IF
END_METHOD

END_FUNCTION_BLOCK

// POUs/model/library/FB_ExecutorTreeSearch
FUNCTION_BLOCK FB_ExecutorTreeSearch
VAR_INPUT
END_VAR
VAR_OUTPUT
END_VAR
VAR
	_observer : InterfaceObserver;
END_VAR

METHOD search : BOOL
VAR_INPUT
	executor : REFERENCE TO FB_Executor;
END_VAR
VAR
	_child_executor  : REFERENCE TO FB_Executor;
	_all_done : BOOL;
END_VAR
_all_done := TRUE;
IF NOT _observer.subscribe_job_directory(executor) THEN
	_all_done := FALSE;
END_IF

// Recursive process if child object exists.
IF executor.children <> 0 THEN
	REPEAT 
		_child_executor REF= executor.children.each_executor;
		IF __ISVALIDREF(_child_executor) THEN
			IF NOT THIS^.search(_child_executor) THEN
				_all_done := FALSE;
			END_IF
		END_IF
	UNTIL
		NOT __ISVALIDREF(_child_executor)
	END_REPEAT	
END_IF
search := _all_done;
END_METHOD

PROPERTY subscriber : InterfaceObserver
SET
_observer := subscriber;
END_SET
END_PROPERTY

END_FUNCTION_BLOCK

// POUs/model/library/FB_ParallelJobContainer
{attribute 'enable_dynamic_creation'}
FUNCTION_BLOCK FB_ParallelJobContainer EXTENDS FB_AbstructContainer
VAR_INPUT
END_VAR
VAR_OUTPUT
END_VAR
VAR
	_initialize :BOOL;
END_VAR

METHOD PROTECTED _append_job : BOOL
VAR_INPUT
	executor	: REFERENCE TO FB_Executor;
END_VAR
VAR
	_parent_future_id :STRING;
END_VAR
IF __ISVALIDREF(executor) AND _num_of_jobs < ParamFuturesLib.MAX_TASK_NUM THEN
	executor.init();
	_num_of_jobs := _num_of_jobs + 1;
	executor.id := UINT_TO_STRING(_num_of_jobs);
	_executors[_num_of_jobs] := ADR(executor);
	IF  __ISVALIDREF(_executor) THEN
		// Propergate task creator object
		_executors[_num_of_jobs]^.job_event_reporter := _executor.job_event_reporter;
		_executors[_num_of_jobs]^.parent_executor REF= _executor;
		_executors[_num_of_jobs]^.upstream_aborting := _executor.upstream_aborting;
		_parent_future_id := _executor.id;
	END_IF
END_IF
END_METHOD

(* This is the generator that iteratively generates references to FB_executor instances*)
METHOD _index_generator_ : UINT
VAR_INST
	_index : UINT;
END_VAR
IF _index > _num_of_jobs THEN
	_index := 0;
ELSE
	_index := _index + 1;
END_IF
_index_generator_ := _index;
END_METHOD

METHOD abort : BOOL // Return TRUE if finish.
VAR
	_all_done : BOOL;
END_VAR
VAR_INST
	_executor : REFERENCE TO FB_Executor;
END_VAR
_all_done := TRUE;
REPEAT
	_executor REF= THIS^.each_executor;
	IF __ISVALIDREF(_executor) THEN
		IF NOT _executor.abort() THEN
			_all_done := FALSE;
		END_IF
	END_IF
UNTIL
	NOT __ISVALIDREF(_executor)
END_REPEAT
abort := _all_done;
END_METHOD

METHOD execute : BOOL // Return TRUE if finish.
VAR_INST
	i :UINT;
	complete_all_task :BOOL;
	wait_for_initilize :BOOL;
END_VAR
IF _num_of_jobs = 0 THEN
	RETURN;
END_IF

complete_all_task := TRUE;
FOR i := 1 TO _num_of_jobs DO
	// Execute all methods
	IF _executors[i]^.current_state < E_FutureExecutionState.finish THEN
		IF NOT _executors[i]^.execute() THEN
			complete_all_task := FALSE;
		END_IF
	END_IF
	
	CASE _executors[i]^.current_state OF 
		E_FutureExecutionState.wait_for_process:
			IF _executors[i]^.ready AND _auto_start THEN
				_executors[i]^.start();
			END_IF
	END_CASE

	_error_id := 0;	
	IF FAILED(_executors[i]^.nErrorID) THEN
		_error_id := _executors[i]^.nErrorID;
	END_IF
END_FOR

current_executing_future := _executors[_num_of_jobs]^.future;

execute := complete_all_task;
END_METHOD

METHOD init : BOOL // Return TRUE if finish.
VAR
	_executor : REFERENCE TO FB_Executor;
	_init_done : BOOL;
END_VAR
_init_done := TRUE;
REPEAT
	_executor REF= THIS^.each_executor;
	IF __ISVALIDREF(_executor) THEN
		_executor.job_event_reporter := _executor.job_event_reporter;
		IF NOT _executor.init() THEN
			_init_done := FALSE;
		END_IF
	END_IF
UNTIL
	NOT __ISVALIDREF(_executor)
END_REPEAT

_error_id := 0;
init := _init_done;
END_METHOD

METHOD quit : BOOL // Return TRUE if finish.
VAR_INST
	i: UINT;
	complete_all_task :BOOL;
END_VAR
complete_all_task := TRUE;
FOR i := 1 TO _num_of_jobs DO
	IF NOT FAILED(_executors[i]^.nErrorID) THEN
		_executors[i]^.execute();
	ELSE
		_error_id := _executors[i]^.nErrorID;
	END_IF
	IF NOT (_executors[i]^.current_state = E_FutureExecutionState.finish) THEN
		complete_all_task := FALSE;	
	END_IF
END_FOR

IF complete_all_task THEN
	_initialize := FALSE;
	quit := TRUE;	
END_IF
END_METHOD

METHOD start : BOOL
VAR
	_all_done : BOOL;
END_VAR
VAR_INST
	_executor : REFERENCE TO FB_Executor;
END_VAR
_all_done := TRUE;
REPEAT
	_executor REF= THIS^.each_executor;
	IF __ISVALIDREF(_executor) THEN
		IF NOT _executor.start() THEN
			_all_done := FALSE;
		END_IF
	END_IF
UNTIL
	NOT __ISVALIDREF(_executor)
END_REPEAT
start := _all_done;
END_METHOD

END_FUNCTION_BLOCK

// POUs/model/library/FB_ParallelJobContainerCreator
FUNCTION_BLOCK FB_ParallelJobContainerCreator IMPLEMENTS InterfaceTaskCreator
VAR_INPUT
END_VAR
VAR_OUTPUT
END_VAR
VAR
END_VAR

{warning 'add method implementation '}
METHOD create_future : InterfaceFuture
VAR_INPUT
	future_name	: STRING;
END_VAR
VAR
	_p_future : POINTER TO FB_ParallelJobContainer;
END_VAR
_p_future := __NEW(FB_ParallelJobContainer);
_p_future^.future_name := future_name;
create_future := _p_future^;
END_METHOD

{warning 'add method implementation '}
METHOD destroy_future : InterfaceFuture
VAR_INPUT
	future	: InterfaceFuture;
END_VAR
VAR
	_p_future : POINTER TO FB_ParallelJobContainer;
END_VAR
IF __QUERYPOINTER(future, _p_future) THEN
	__DELETE(_p_future);
	IF _p_future = 0  THEN
		destroy_future := 0;
	END_IF
END_IF
END_METHOD

END_FUNCTION_BLOCK

// POUs/model/library/FB_ParallelQueueJobContainer
{attribute 'enable_dynamic_creation'}
FUNCTION_BLOCK FB_ParallelQueueJobContainer EXTENDS FB_AbstructContainer
VAR_INPUT
END_VAR
VAR_OUTPUT
END_VAR
VAR
END_VAR
VAR PERSISTENT
	_serial	: ULINT := 1;
END_VAR

METHOD PROTECTED _append_job : BOOL
VAR_INPUT
	executor	: REFERENCE TO FB_Executor;
END_VAR
VAR
	future_order_number: INT;
	_parent_future_id: STRING;
	i: 	UINT := 1;
END_VAR
//Set buffer index
IF _num_of_jobs < ParamFuturesLib.MAX_TASK_NUM THEN
	i := 1;
	WHILE _executors[i] <> 0 DO
		i := i + 1;
	END_WHILE

	// Spawn new task with specified future
	executor.init();
	_executors[i] := ADR(executor);
	
	// Get parent task id
	IF  __ISVALIDREF(_executor) THEN
		_executors[i]^.job_event_reporter := _executor.job_event_reporter;
		_executors[i]^.parent_executor REF= _executor;
		_executors[i]^.upstream_aborting := _executor.upstream_aborting;
		_parent_future_id := _executor.id;
	END_IF
	_executors[i]^.id := ULINT_TO_STRING(_serial);
	_serial := _serial + 1;
	IF _serial = 16#FFFFFFFFFFFFFFFF THEN
		_serial := 0;
	END_IF
	_num_of_jobs := _num_of_jobs + 1;
END_IF
END_METHOD

(* This is the generator that iteratively generates references to FB_executor instances*)
METHOD _index_generator_ : UINT;
VAR_INPUT
END_VAR
VAR_INST
	_init	: BOOL := FALSE;
	_current_order_number : UINT; // Represent order number of iteration
	_index: UINT;
END_VAR
IF NOT _init THEN
	_current_order_number := 0;
	_index := 1;
	_index_generator_ := 0;
	_init := TRUE;
END_IF

IF _num_of_jobs = 0 THEN
	RETURN;
END_IF


IF _current_order_number >= _num_of_jobs OR _index > ParamFuturesLib.MAX_TASK_NUM THEN
	_init := FALSE;
END_IF

IF _init THEN
	WHILE _index < ParamFuturesLib.MAX_TASK_NUM AND _executors[_index] = 0 DO
		_index := _index + 1;
	END_WHILE
	IF _executors[_index] <> 0 THEN
		_index_generator_ := _index;
	ELSE
		_index_generator_ := 0;
	END_IF
	_current_order_number := _current_order_number + 1;
	_index := _index + 1;
ELSE
	_index_generator_ := 0;
END_IF
END_METHOD

METHOD abort : BOOL // Return TRUE if finish.
VAR
	_all_done : BOOL;
END_VAR
VAR_INST
	_executor : REFERENCE TO FB_Executor;
END_VAR
_all_done := TRUE;
REPEAT
	_executor REF= THIS^.each_executor;
	IF __ISVALIDREF(_executor) THEN
		IF NOT _executor.abort() THEN
			_all_done := FALSE;
		END_IF
	END_IF
UNTIL
	NOT __ISVALIDREF(_executor)
END_REPEAT
abort := _all_done;
END_METHOD

METHOD execute : BOOL // Return TRUE if finish.
VAR
	_head : BOOL;
	_future_id :UINT;
	i: UINT;
END_VAR
execute := FALSE;

IF _num_of_jobs = 0 THEN
	RETURN;
END_IF

REPEAT
	// キューインされたFB_executorインスタンスを順に取り出すイテレータ。_endがTRUEになれば全て取り出し完了。_headは先頭のみtrueになる。
	i := _index_generator_();
	IF i > 0 THEN
		IF _executors[i]^.execute() THEN
			IF _executors[i]^.reset(FALSE) THEN
				IF _executors[i]^.persistent_job THEN
					_executors[i] := 0;
				ELSE
					__DELETE(_executors[i]);
				END_IF
				_num_of_jobs := _num_of_jobs - 1;
			END_IF
			execute := _num_of_jobs = 0 AND NOT _continuous_mode;
		ELSE
			CASE _executors[i]^.current_state OF
				E_FutureExecutionState.idle:
					_executors[i]^.init();
				E_FutureExecutionState.wait_for_process:
					_executors[i]^.start();
				E_FutureExecutionState.init, E_FutureExecutionState.process, E_FutureExecutionState.quit:
					IF 	_executors[i]^.current_state = E_FutureExecutionState.process THEN
						// Report total futures
						current_executing_future := _executors[i]^.future;						
					END_IF
			END_CASE
			_error_id := _executors[i]^.nErrorID;
		END_IF
	END_IF
UNTIL
	i = 0
END_REPEAT
END_METHOD

METHOD init : BOOL // Return TRUE if finish.
VAR
	_executor : REFERENCE TO FB_Executor;
	_init_done : BOOL;
END_VAR
_init_done := TRUE;
REPEAT
	_executor REF= THIS^.each_executor;
	IF __ISVALIDREF(_executor) THEN
		_executor.job_event_reporter := _executor.job_event_reporter;
		IF NOT _executor.init() THEN
			_init_done := FALSE;
		END_IF
	END_IF
UNTIL
	NOT __ISVALIDREF(_executor)
END_REPEAT

_error_id := 0;
init := _init_done;
END_METHOD

METHOD start : BOOL
VAR
	_all_done : BOOL;
END_VAR
VAR_INST
	_executor : REFERENCE TO FB_Executor;
END_VAR
_all_done := TRUE;
REPEAT
	_executor REF= THIS^.each_executor;
	IF __ISVALIDREF(_executor) THEN
		IF NOT _executor.start() AND _executor.ready THEN
			_all_done := FALSE;
		END_IF
	END_IF
UNTIL
	NOT __ISVALIDREF(_executor)
END_REPEAT
start := _all_done;
END_METHOD

END_FUNCTION_BLOCK

// POUs/model/library/FB_ParallelQueueJobContainerCreator
FUNCTION_BLOCK FB_ParallelQueueJobContainerCreator IMPLEMENTS InterfaceTaskCreator
VAR_INPUT
END_VAR
VAR_OUTPUT
END_VAR
VAR
END_VAR

{warning 'add method implementation '}
METHOD create_future : InterfaceFuture
VAR_INPUT
	future_name	: STRING;
END_VAR
VAR
	_p_future : POINTER TO FB_ParallelQueueJobContainer;
END_VAR
_p_future := __NEW(FB_ParallelQueueJobContainer);
_p_future^.future_name := future_name;
create_future := _p_future^;
END_METHOD

{warning 'add method implementation '}
METHOD destroy_future : InterfaceFuture
VAR_INPUT
	future	: InterfaceFuture;
END_VAR
VAR
	_p_future : POINTER TO FB_ParallelQueueJobContainer;
END_VAR
IF __QUERYPOINTER(future, _p_future) THEN
	__DELETE(_p_future);
	IF _p_future = 0  THEN
		destroy_future := 0;
	END_IF
END_IF
END_METHOD

END_FUNCTION_BLOCK

// POUs/model/library/FB_QueueJobContainer
{attribute 'enable_dynamic_creation'}
FUNCTION_BLOCK FB_QueueJobContainer EXTENDS FB_AbstructContainer
VAR_INPUT
END_VAR
VAR_OUTPUT
END_VAR
VAR
	_current_executing_job : REFERENCE TO FB_Executor;
	nWriteIndex: 	UINT := 1;
	nReadIndex: 	UINT := 1;
END_VAR
VAR PERSISTENT
	_serial	: ULINT := 1;
END_VAR

METHOD PROTECTED _append_job : BOOL
VAR_INPUT
	executor	: REFERENCE TO FB_Executor;
END_VAR
VAR_INST
	carry_flag:		BOOL;
END_VAR
//Set buffer index
IF __ISVALIDREF(executor) AND _num_of_jobs < ParamFuturesLib.MAX_TASK_NUM THEN
	executor.init();
	// Spawn new task with specified feature
	_executors[nWriteIndex] := ADR(executor);

	// Get parent tssk id
	IF  __ISVALIDREF(_executor) THEN
		_executors[nWriteIndex]^.job_event_reporter := _executor.job_event_reporter;
		_executors[nWriteIndex]^.parent_executor REF= _executor;
		_executors[nWriteIndex]^.upstream_aborting := _executor.upstream_aborting;
	END_IF

	// Set my task ID
	_executors[nWriteIndex]^.id := ULINT_TO_STRING(_serial);
	
	// generate new serial number
	IF _serial = 16#FFFFFFFFFFFFFFFF THEN
		_serial := 0;
	END_IF
	_serial := _serial + 1;


	nWriteIndex := nWriteIndex + 1;
	IF nWriteIndex > ParamFuturesLib.MAX_TASK_NUM THEN
		nWriteIndex := 1;
	END_IF
	
	IF nWriteIndex = nReadIndex AND _num_of_jobs = ParamFuturesLib.MAX_TASK_NUM - 1 THEN 
		carry_flag := TRUE;
	END_IF

	// calculate order number of executing futures by queue address
	IF carry_flag THEN
		_num_of_jobs := ParamFuturesLib.MAX_TASK_NUM;
		carry_flag := FALSE;
	ELSIF nWriteIndex >= nReadIndex THEN
		_num_of_jobs := nWriteIndex - nReadIndex;
	ELSE
		_num_of_jobs := ParamFuturesLib.MAX_TASK_NUM - nReadIndex + nWriteIndex;
	END_IF

END_IF
END_METHOD

(* This is the generator that iteratively generates references to FB_executor instances*)
METHOD _index_generator_ : UINT;
VAR_INST
	_init	: BOOL := FALSE;
	_index :UINT;
	_current_order_number : DINT;
	_carry_flag : BOOL;
END_VAR
IF NOT _init THEN
	_carry_flag := FALSE;
	_index := nReadIndex;
	_init := TRUE;
END_IF

// calculate order number of executing futures by queue address
IF _num_of_jobs = 0 THEN
	_current_order_number := 0;
ELSIF _carry_flag THEN // 
	_current_order_number := ParamFuturesLib.MAX_TASK_NUM;
ELSIF nWriteIndex > nReadIndex THEN // Normal case
	_current_order_number := _index - nReadIndex + 1;
ELSE // 
	_current_order_number := _index - nReadIndex + 1;
	IF _current_order_number < 0 THEN
		_current_order_number := _current_order_number + ParamFuturesLib.MAX_TASK_NUM;
	END_IF
	IF _current_order_number = ParamFuturesLib.MAX_TASK_NUM - 1 THEN
		_carry_flag := TRUE;
	END_IF
END_IF


_index_generator_ := _index;

//Set buffer index
IF _num_of_jobs = 0 OR _num_of_jobs < _current_order_number THEN
	_init := FALSE;
END_IF

IF NOT _init THEN
	_index_generator_ := 0;
END_IF

IF _init THEN
	_index := _index + 1;
	IF _index > ParamFuturesLib.MAX_TASK_NUM THEN
		_index := 1;
	END_IF
END_IF
END_METHOD

METHOD abort : BOOL // Return TRUE if finish.
IF __ISVALIDREF(_current_executing_job) THEN
	abort := _current_executing_job.abort();
ELSE
	abort := TRUE;
END_IF
END_METHOD

METHOD dequeue : POINTER TO FB_Executor;
VAR_INPUT
END_VAR
//Set buffer index
IF _num_of_jobs > 0 THEN
	dequeue := _executors[nReadIndex];
	nReadIndex := nReadIndex + 1;
	IF nReadIndex > ParamFuturesLib.MAX_TASK_NUM THEN
		nReadIndex := 1;
	END_IF
	// calculate order number of executing futures by queue address
	IF nWriteIndex >= nReadIndex THEN
		_num_of_jobs := nWriteIndex - nReadIndex;
	ELSE
		_num_of_jobs := ParamFuturesLib.MAX_TASK_NUM - nReadIndex + nWriteIndex;
	END_IF
ELSE
	dequeue := 0;
END_IF
END_METHOD

METHOD execute : BOOL // Return TRUE if finish.
VAR
	_head : BOOL;
	_execution_complete :BOOL; 
	_future_id :UINT;
	complete_last_proess :BOOL := FALSE;
	i: UINT;
	_finish_delay : TON;
	_executor : POINTER TO FB_Executor;
END_VAR
complete_last_proess := FALSE;

//IF _total_futures = 0 THEN
//	RETURN;
//END_IF

_head := TRUE;
REPEAT
	// キューインされたFB_executorインスタンスを順に取り出すイテレータ。_endがTRUEになれば全て取り出し完了。_headは先頭のみtrueになる。
	i := THIS^._index_generator_();
	
	IF i > 0 THEN
		_executor := _executors[i];
		_execution_complete := _executor^.execute();
		
		CASE _executor^.current_state OF
			E_FutureExecutionState.idle:
				_executor^.init();
			E_FutureExecutionState.wait_for_process:
				IF _executor^.ready AND (complete_last_proess OR _head) AND _auto_start THEN
					_executor^.start();
					_current_executing_job REF= _executor^;
				END_IF
		END_CASE
		
		complete_last_proess := _executor^.done;	

		_error_id := _executor^.nErrorID;
		
		IF _execution_complete THEN
			IF _head THEN
				// キューの先頭がfinish状態になれば取り出してキューから削除する
				IF _executor^.reset(FALSE) THEN
					THIS^.dequeue();
					IF NOT _executor^.persistent_job THEN
						__DELETE(_executor);
					END_IF
				END_IF
			END_IF		
		END_IF
	ELSIF  _execution_complete THEN
		execute := NOT _continuous_mode;
	END_IF
	_head := FALSE;
UNTIL
	i = 0
END_REPEAT;
END_METHOD

METHOD init : BOOL // Return TRUE if finish.
VAR
	_executor : REFERENCE TO FB_Executor;
	_init_done : BOOL;
END_VAR
_init_done := TRUE;
REPEAT
	_executor REF= THIS^.each_executor;
	IF __ISVALIDREF(_executor) THEN
		_executor.job_event_reporter := _executor.job_event_reporter;
		IF NOT _executor.init() THEN
			_init_done := FALSE;
		END_IF
	END_IF
UNTIL
	NOT __ISVALIDREF(_executor)
END_REPEAT

_current_executing_job REF= 0;
_error_id := 0;
init := _init_done;
END_METHOD

METHOD start : BOOL
VAR
	_all_done : BOOL;
END_VAR
VAR_INST
	_executor : REFERENCE TO FB_Executor;
END_VAR
IF __ISVALIDREF(_current_executing_job) THEN
	IF _current_executing_job.ready THEN
		start := _current_executing_job.start();
	ELSE
		start := TRUE;	
	END_IF
ELSE
	start := TRUE;
END_IF
END_METHOD

END_FUNCTION_BLOCK

// POUs/model/library/FB_QueueJobContainerCreator
FUNCTION_BLOCK FB_QueueJobContainerCreator IMPLEMENTS InterfaceTaskCreator
VAR_INPUT
END_VAR
VAR_OUTPUT
END_VAR
VAR
END_VAR

{warning 'add method implementation '}
METHOD create_future : InterfaceFuture
VAR_INPUT
	future_name	: STRING;
END_VAR
VAR
	_p_future : POINTER TO FB_QueueJobContainer;
END_VAR
_p_future := __NEW(FB_QueueJobContainer);
_p_future^.future_name := future_name;
create_future := _p_future^;
END_METHOD

{warning 'add method implementation '}
METHOD destroy_future : InterfaceFuture
VAR_INPUT
	future	: InterfaceFuture;
END_VAR
VAR
	_p_future : POINTER TO FB_QueueJobContainer;
END_VAR
IF __QUERYPOINTER(future, _p_future) THEN
	__DELETE(_p_future);
	IF _p_future = 0  THEN
		destroy_future := 0;
	END_IF
END_IF
END_METHOD

END_FUNCTION_BLOCK

// POUs/MAIN
PROGRAM MAIN
VAR
	_state :UINT;
	actual_job : REFERENCE TO FB_Executor;
	executor: FB_Executor; // main Executor
	
	_child_executor : REFERENCE TO FB_Executor;
	
	task_blink_1 : FutureTimerBlink;
	task_blink_2 : FutureTimerBlink;
	task_count_1 : FutureCounterBlink;
	task_count_2 : FutureCounterBlink;

	future_counter_creator : FutureCounterBlinkCreator;
	future_timer_creator : FutureTimerBlinkCreator;

	
	component1_in : BOOL;
	component1_out : BOOL;
	component2_in : BOOL;
	component2_out : BOOL;
	component3_in : BOOL;
	component3_out : BOOL;
	component4_in : BOOL;
	component4_out : BOOL;

	
	// Dynamic instance use
	_future: InterfaceFuture;
	_container : InterfaceContainer;
	
	job_create_switch : ARRAY[1..4] OF BOOL;
	execution_step: STRING;
	resume: BOOL;
	abort: BOOL;
	reset : BOOL;
	task_info : __SYSTEM.VAR_INFO;
	
	fbObserver : FB_observer;
	fbJobTreeSearch : FB_ExecutorTreeSearch;
	
	end_of_manual: BOOL;
	init :BOOL;
	test_executor : POINTER TO FB_BatchJobContainer;
	
	future_timer : FutureTimerBlink;
	future_counter : FutureCounterBlink;
	
	_monitor_job : REFERENCE TO FB_Executor;
	_monitor_count_blinker : POINTER TO FutureCounterBlink;
	_monitor_time_blinker : POINTER TO FutureTimerBlink;
	
	_job_debug_monitoring : FB_Executor;
	
END_VAR

IF NOT init THEN
	//executor.job_event_reporter := fbObserver;
	init := TRUE;
	executor.id := 'ROOT';
	executor.upstream_aborting := FALSE;
	executor.create_container(ContainerType.PARALLEL_QUEUE,'BASE');
	executor.continuous_mode := TRUE;
	executor.job_event_reporter := fbObserver;
	//actual_job REF= executor.children.create_container(ContainerType.QUEUE, 'Batch Container');
	//actual_job.continuous_mode := TRUE;
END_IF

IF abort THEN
	executor.abort();
END_IF

executor.execute();

IF executor.ready THEN
	executor.start();
END_IF

IF resume THEN
	IF executor.error_reset() THEN
		IF executor.resume() THEN
			resume := FALSE;
		END_IF
	END_IF
END_IF



CASE _state OF
	0:
		_child_executor REF= executor.children.create_container(ContainerType.PARALLEL_QUEUE, 'Parallel Container');
		// Static instances
		task_blink_1.set_parameter(T#5S, component1_out);
		task_blink_1.future_name := 'Button 1 blink';
		task_blink_2.set_parameter(T#3S, component2_out);
		task_blink_2.future_name := 'Button 2 blink';
		task_count_1.set_parameter(3, component3_in,component3_out);
		task_count_1.future_name := 'Button 3 count';
		task_count_2.set_parameter(5, component4_in, component4_out);
		task_count_2.error_test := FALSE;
		task_count_2.future_name := 'Button 4 count';
		
		_child_executor.children.spawn_job(task_blink_1);
		_child_executor.children.spawn_job(task_blink_2);
		_child_executor.children.spawn_job(task_count_1);
		_child_executor.children.spawn_job(task_count_2);
		__QUERYPOINTER(_child_executor.children,test_executor);
		
		// dynamic instances		
		//_child_executor REF= actual_job.children.create_container(ContainerType.PARALLEL, 'Dynamic parallel tasks');
		
		future_counter_creator.set_parameter(2, component3_in, component3_out);
		_child_executor.children.create_job(future_counter_creator, 'Dynamic job : Count-1');	
		
		future_counter_creator.set_parameter(5, component4_in, component4_out);
		_child_executor.children.create_job(future_counter_creator, 'Dynamic job : Count-2');

		future_counter_creator.set_parameter(2,component3_in, component3_out);
		_child_executor.children.create_job(future_counter_creator, 'Dynamic job : Counter3');

		future_counter_creator.set_parameter(2, component3_in, component3_out);
		_child_executor.children.create_job(future_counter_creator, 'Dynamic job : Counter4'); // 同時実行でなければ同じFutureオブジェクトを使いまわせる
		future_counter_creator.set_parameter(2, component4_in, component4_out);
		_child_executor.children.create_job(future_counter_creator, 'Dynamic job : Counter5');
		
		// Report 'executor' job directory
		fbJobTreeSearch.subscriber := fbObserver;
		fbJobTreeSearch.search(executor);
			
		_state := 1;
	1:
		// シーケンス制御
		IF _child_executor.done THEN
			_state := 3;
		END_IF
	2:
		_state := 3;			
	3:
		
		IF job_create_switch[1] THEN
			future_timer_creator.set_parameter(T#5S, component1_out);
			future_timer_creator.set_options(FALSE);
			_monitor_job REF= executor.children.create_job(future_timer_creator, 'Button 1 Time blink 5s');
			IF NOT  __QUERYPOINTER(_monitor_job.future, _monitor_count_blinker) THEN
				_monitor_count_blinker := 0;
			END_IF
			IF NOT __QUERYPOINTER(_monitor_job.future, _monitor_time_blinker)  THEN
				_monitor_time_blinker := 0;
			END_IF
			job_create_switch[1] := FALSE;
		
		ELSIF job_create_switch[2] THEN
			future_timer_creator.set_parameter(T#3S, component2_out);
			future_timer_creator.set_options(FALSE);
			_monitor_job REF= executor.children.create_job(future_timer_creator, 'Button 2 Time blink 3s');
			IF NOT  __QUERYPOINTER(_monitor_job.future, _monitor_count_blinker) THEN
				_monitor_count_blinker := 0;
			END_IF
			IF NOT __QUERYPOINTER(_monitor_job.future, _monitor_time_blinker)  THEN
				_monitor_time_blinker := 0;
			END_IF
			job_create_switch[2] := FALSE;
		
		ELSIF  job_create_switch[3] THEN
			job_create_switch[3] := FALSE;
			future_counter_creator.set_parameter(2, component3_in, component3_out);
			future_counter_creator.set_options(FALSE);
			_monitor_job REF= executor.children.create_job(future_counter_creator, 'Dynamic job : Counter6');
			IF NOT  __QUERYPOINTER(_monitor_job.future, _monitor_count_blinker) THEN
				_monitor_count_blinker := 0;
			END_IF
			IF NOT __QUERYPOINTER(_monitor_job.future, _monitor_time_blinker)  THEN
				_monitor_time_blinker := 0;
			END_IF
			job_create_switch[3] := FALSE;
		ELSIF  job_create_switch[4] THEN
			job_create_switch[4] := FALSE;
			future_counter_creator.set_parameter(4, component4_in, component4_out);
			future_counter_creator.set_options(TRUE);
			_monitor_job REF= executor.children.create_job(future_counter_creator, 'Dynamic job : Counter7');
			IF NOT  __QUERYPOINTER(_monitor_job.future, _monitor_count_blinker) THEN
				_monitor_count_blinker := 0;
			END_IF
			IF NOT __QUERYPOINTER(_monitor_job.future, _monitor_time_blinker)  THEN
				_monitor_time_blinker := 0;
			END_IF
			job_create_switch[4] := FALSE;
		
		END_IF
		IF reset THEN
			executor.quit();
			_state := 4;
		END_IF
	4:
		_state := 0;
		
END_CASE

MEMCPY(ADR(_job_debug_monitoring), ADR(_child_executor), SIZEOF(_job_debug_monitoring));

IF reset AND NOT executor.busy THEN
	IF executor.children.reset(TRUE) THEN
		reset := FALSE;
	END_IF
END_IF

END_PROGRAM

// VISUs/Visualization
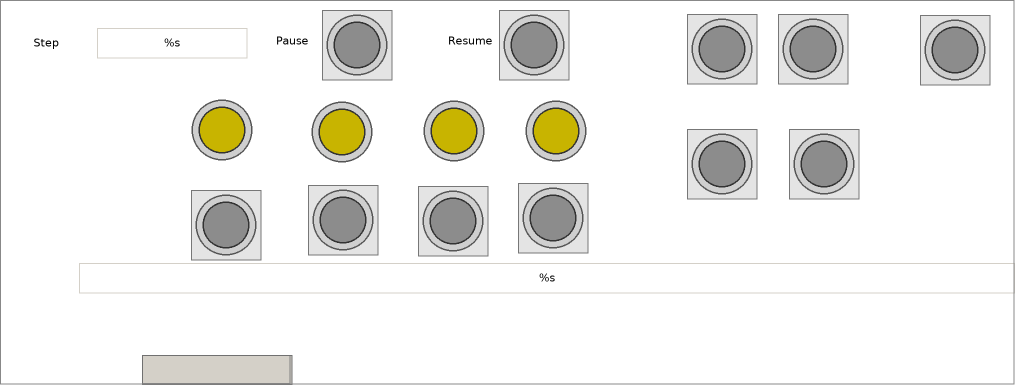
VISUALIZATION Visualization  // 1015x385
    PushSwitch (191,190 70x70), variable: MAIN.component1_in, behaviour: TAP, style: Switch-PushSwitch-Gray
    PushSwitch (308,185 70x70), variable: MAIN.component2_in, behaviour: TAP, style: Switch-PushSwitch-Gray
    PushSwitch (418,186 70x70), variable: MAIN.component3_in, behaviour: TAP, style: Switch-PushSwitch-Gray
    PushSwitch (518,183 70x70), variable: MAIN.component4_in, behaviour: TAP, style: Switch-PushSwitch-Gray
    Lamp1 (187,95 70x70), variable: MAIN.component1_out, style: Lamp-Lamp1-Yellow
    Lamp1 (307,97 70x70), variable: MAIN.component2_out, style: Lamp-Lamp1-Yellow
    Lamp1 (419,96 70x70), variable: MAIN.component3_out, style: Lamp-Lamp1-Yellow
    Lamp1 (521,96 70x70), variable: MAIN.component4_out, style: Lamp-Lamp1-Yellow
    Textfield (97,28 150x30), "%s", text variable: MAIN.execution_step
    PushSwitch (322,10 70x70), variable: MAIN.abort, behaviour: TAP, style: Switch-PushSwitch-Gray
    PushSwitch (499,10 70x70), variable: MAIN.resume, behaviour: TOGGLE, style: Switch-PushSwitch-Gray
    Label (259,26 67x30), "Pause"
    Label (437,26 67x30), "Resume"
    Label (13,28 67x30), "Step"
    PushSwitch (687,14 70x70), variable: MAIN.job_create_switch[1], behaviour: TOGGLE, style: Switch-PushSwitch-Gray
    PushSwitch (778,14 70x70), variable: MAIN.job_create_switch[2], behaviour: TOGGLE, style: Switch-PushSwitch-Gray
    PushSwitch (687,129 70x70), variable: MAIN.job_create_switch[3], behaviour: TOGGLE, style: Switch-PushSwitch-Gray
    PushSwitch (789,129 70x70), variable: MAIN.job_create_switch[4], behaviour: TOGGLE, style: Switch-PushSwitch-Gray
    PushSwitch (920,15 70x70), variable: MAIN.reset, behaviour: TOGGLE, style: Switch-PushSwitch-Gray
    Textfield (79,263 936x30), "%s", text variable: MAIN.fbObserver.text
    Button (142,355 150x30)
        OnMouseDown:  Assign=Visualization_1, Type=Assignment
END_VISUALIZATION

// VISUs/Visualization_1
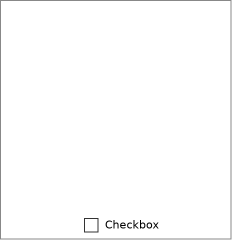
VISUALIZATION Visualization_1  // 232x240
    Checkbox (82,210 150x30), "Checkbox"
END_VISUALIZATION
